{attribute 'GeneratedUsingTerminal: EK1100-0000-0018'}
{attribute addProperty BoxType "EK1100-0000-0018"}
{attribute addProperty Id "Beckhoff_AT2xxxEK1122Beckhoff_AT2xxxEK1122_5BEE8A185530A_0059_AT2000_5250_0018AT2000_33A3DF1B80"}
{attribute addProperty CRC "2622014049"}
{attribute addProperty Size "5610"}
TYPE Beckhoff_AT1xxx_9C48C261 EXTENDS EK1100_1FC0878B :
STRUCT
	{attribute addProperty Name "Beckhoff_AT2xxxEK1122"}
	{attribute addProperty PreviousPort "Beckhoff AT1xxx : B"}
	Beckhoff_AT2xxxEK1122 : Beckhoff_AT2xxxEK1122_5BEE8A18;
	{attribute addProperty Name "A_0059_AT2000_5250_0018"}
	{attribute addProperty PreviousPort "Beckhoff AT2xxxEK1122 : C"}
	A_0059_AT2000_5250_0018 : AT2000_33A3DF1B;
END_STRUCT
END_TYPE

(* stored: Version 1.2.0.0, ProductVersion 3.1.4024.9
   DUT Beckhoff_AT1xxx_9C48C261: Id {089403bb-12f4-47ea-8ee4-94ff1bc16123} *)
